FUNCTION_BLOCK FB_ImageAquire EXTENDS FB_VisionCameraBase
VAR
	_Image			 : ITcVnImage;
	_ImageAvailable	 : BOOL;
	ipImageInDisplay : ITcVnDisplayableImage;
END_VAR

PROPERTY Image : ITcVnImage
GET
Image := _Image;
_ImageAvailable := FALSE;
END_GET
END_PROPERTY

PROPERTY ImageAvailable : BOOL
GET
ImageAvailable := _ImageAvailable;
END_GET
END_PROPERTY

METHOD PUBLIC  ProcessImage
hr := F_VN_CopyIntoDisplayableImage(ipImageIn,ipImageInDisplay,S_OK);


hr := F_VN_CopyImage(ipImageIn,_Image, S_OK);
_ImageAvailable := TRUE;
END_METHOD

END_FUNCTION_BLOCK

(* stored: Version 1.1.0.1, ProductVersion 3.1.4024.12
   POU FB_ImageAquire: Id {d1d4ab92-b3c1-4cac-ab3a-010aa8210778}, SpecialFunc None
   Property Image: Id {10d4dd17-8a58-4b1c-8f0d-16512446eea3}
   Get Get: Id {debe11ac-9225-4cab-bcb2-b378dacbf1ea}
   Property ImageAvailable: Id {cf6a288e-379c-4676-a5c8-a4e2f6f5445c}
   Get Get: Id {5dae1fd6-ec7e-4d0c-8413-f404f7b7d352}
   Method ProcessImage: Id {31a1b0a1-87b1-464c-a92d-a4586f368e25} *)
